// TIA Portal V18 export
FUNCTION_BLOCK "LAxisGroupBasics_AxisGroupBasics_Grp1"   // FB5, SCL
{ S7_Optimized_Access := 'TRUE' }
// stored: MemoryReserve 100, SetENOAutomatically false
   VAR_INPUT
      powerEnableAll : Bool;   // MC_Power: 0: Disable all axes/ 1: Enable all axes
      homeExecuteAll : Bool;   // MC_Home: Start job for all axes with positive edge
      resetExecuteAll : Bool;   // MC_Reset: Start job for all axes with positive edge
      restartAll : Bool;   // 0: Acknowledgment of queued technology alarms / 1: Reinitialization of the technology object and acknowledgment of pending technology alarms
      haltExecuteAll : Bool;   // MC_Halt: Start job for all axes with positive edge
   END_VAR
   VAR_OUTPUT
      powerStatusGroup : Bool;   // MC_Power: 0: At least one Technology object disabled / 1: All Technology objects enabled
      homingStatusGroup : Bool;   // MC_Home: 0: At least one Technology object
      busy : Bool;   // Job is running
      done : Bool;   // All active jobs done
      commandAborted : Bool;   // At least one command was aborted
      error : Bool;   // An error occurred during execution of the job. The job is rejected. The cause of the error can be found in the "Status" parameter.
      status : Word;   // Status information
      diagnostics : "LAxisGroupBasics_typeDiagnostics";   // Diagnostics information
   END_VAR
   VAR_IN_OUT
      axisGroupBasicsData : Array[*] of "LAxisGroupBasics_typeAxisGroupBasicsData";   // Axis data
   END_VAR
   VAR
      instAxisBasics : Array[#LOWER_LIMIT_AXES_ARRAY..#UPPER_LIMIT_AXES_ARRAY] of "LAxisBasics_AxisBasics";
      statErrorIndexOld { ExternalAccessible := 'False'; ExternalVisible := 'False'; ExternalWritable := 'False'} : DInt;   // Flag for saving error index
      statAxisBasicsStatusOld { ExternalAccessible := 'False'; ExternalVisible := 'False'; ExternalWritable := 'False'} : Word;   // Flag for saving LAxisBasics status
      statAxisBasicsSubfunctionStatusOld { ExternalAccessible := 'False'; ExternalVisible := 'False'; ExternalWritable := 'False'} : Word;   // Flag for savin LAxisBasics subfunction status
   END_VAR
   VAR_TEMP
      tempAxisArrayLowerBound : DInt;   // Start index of axes array
      tempAxisArrayUpperBound : DInt;   // End index of axes array
      tempIndex : DInt;   // index counter
      tempDateTimeRetVal : Int;   // date time return value
      tempError : Bool;   // temporary error bit
      tempBusy : Bool;   // temporary busy bit
      tempDone : Bool;   // temporary done bit
      tempCmdAborted : Bool;   // temporary command aborted bit
      tempPowerStatusGroup : Bool;   // temporary power status group bit
      tempHomingStatusGroup : Bool;   // temporary homing status group bit
      tempFirstErrorIndex : DInt;   // index at which first error occured
      tempNewError : Bool;   // new error occured in this cycle
   END_VAR
   VAR CONSTANT
      LOWER_LIMIT_AXES_ARRAY : DInt := 0;   // Start index of axes array needs to be adapted to real array dimensons
      UPPER_LIMIT_AXES_ARRAY : DInt := 4;   // End index of axes array needs to be adapted to real array dimensions
      STATUS_INCORRECT_ARRAY_CONSTANTS : Word := 16#8310;   // status value incorrect array constants
      STATUS_ERR_SYSTEMFUNCTION : Word := 16#8600;   // status value error LAxisBasics
      STATUS_ACTIVE : Word := 16#7002;   // status value active
      STATUS_INACTIVE : Word := 16#7000;   // status value inactive
      DEFAULT_DATE_TIME : Date_And_Time := DT#1990-01-01-00:00:00;   // date and time default value
      DEFAULT_STATUS : Word := 16#0;   // status value default
      ADD_VALUE1_DEFAULT : Int := 0;   // additional value 1 default
      ADD_VALUE2_DEFAULT : Word;   // additional value 2 default
      EMPTY : DInt := -1;   // empty
   END_VAR
BEGIN
   //=============================================================================
   //SIEMENS AG
   //(c)Copyright 2016 All Rights Reserved
   //-----------------------------------------------------------------------------
   //Library:       Axis Basics
   //Tested with:   S7-1500T V3.0
   //Engineering:   TIA Portal V18
   //Restrictions:  Motion Control Library V7.0
   //Requirements:  S7-1500(T)
   //Functionality: Basic axis group control and data collection
   //-----------------------------------------------------------------------------
   //Change log table:
   //Version  Date       Expert in charge Changes applied
   //01.00.00 01.08.2023 FrJu             First released version
   //=============================================================================

   REGION Axis array checks
       //Check Array boundaries of axis array
       #tempAxisArrayUpperBound := UPPER_BOUND(ARR := #axisGroupBasicsData, DIM := 1);
       #tempAxisArrayLowerBound := LOWER_BOUND(ARR := #axisGroupBasicsData, DIM := 1);

       //Check if number of axes/array length is matching - output error and return if values are not matching
       IF #tempAxisArrayUpperBound <> #UPPER_LIMIT_AXES_ARRAY
           OR #tempAxisArrayLowerBound <> #LOWER_LIMIT_AXES_ARRAY THEN

           #error := TRUE;
           #status := #diagnostics.status := #STATUS_INCORRECT_ARRAY_CONSTANTS;

           RETURN;
       END_IF;
   END_REGION

   REGION Initialize values
       //initialize values
       #tempError := FALSE;
       #tempBusy := FALSE;
       #tempDone := FALSE;
       #tempPowerStatusGroup := TRUE;
       #tempHomingStatusGroup := TRUE;
       #tempFirstErrorIndex := #EMPTY;
       #tempCmdAborted := FAlSE;
   END_REGION

   REGION Axes operation loop
       //Loop through all instances of LAxisBasics and execute commands
       FOR #tempIndex := #tempAxisArrayLowerBound TO #tempAxisArrayUpperBound DO

           REGION Call AxisBasics
               //Call LAxisBasics_AxisBasics
               #instAxisBasics[#tempIndex](axis := #axisGroupBasicsData[#tempIndex].axis,
                                           powerEnable := #axisGroupBasicsData[#tempIndex].axisBasicsData.axisControl.axisControlCommand.powerEnable OR #powerEnableAll,
                                           powerStartMode := #axisGroupBasicsData[#tempIndex].axisBasicsData.axisControl.axisControlCommand.powerStartMode,
                                           powerStopMode := #axisGroupBasicsData[#tempIndex].axisBasicsData.axisControl.axisControlCommand.powerStopMode,
                                           resetExecute := #axisGroupBasicsData[#tempIndex].axisBasicsData.axisControl.axisControlCommand.resetExecute OR #resetExecuteAll,
                                           resetRestart := #axisGroupBasicsData[#tempIndex].axisBasicsData.axisControl.axisControlCommand.resetRestart OR #restartAll,
                                           homeExecute := #axisGroupBasicsData[#tempIndex].axisBasicsData.axisControl.axisControlCommand.homeExecute OR #homeExecuteAll,
                                           homePosition := #axisGroupBasicsData[#tempIndex].axisBasicsData.axisControl.axisControlCommand.homePosition,
                                           homeMode := #axisGroupBasicsData[#tempIndex].axisBasicsData.axisControl.axisControlCommand.homeMode,
                                           jogForward := #axisGroupBasicsData[#tempIndex].axisBasicsData.axisControl.axisControlCommand.jogForward,
                                           jogBackward := #axisGroupBasicsData[#tempIndex].axisBasicsData.axisControl.axisControlCommand.jogBackward,
                                           jogVelocity := #axisGroupBasicsData[#tempIndex].axisBasicsData.axisControl.axisControlCommand.jogVelocity,
                                           jogAcceleration := #axisGroupBasicsData[#tempIndex].axisBasicsData.axisControl.axisControlCommand.jogAcceleration,
                                           jogDeceleration := #axisGroupBasicsData[#tempIndex].axisBasicsData.axisControl.axisControlCommand.jogDeceleration,
                                           jogJerk := #axisGroupBasicsData[#tempIndex].axisBasicsData.axisControl.axisControlCommand.jogJerk,
                                           jogPositionControlled := #axisGroupBasicsData[#tempIndex].axisBasicsData.axisControl.axisControlCommand.jogPositionControlled,
                                           moveAbsExecute := #axisGroupBasicsData[#tempIndex].axisBasicsData.axisControl.axisControlCommand.moveAbsExecute,
                                           moveRelExecute := #axisGroupBasicsData[#tempIndex].axisBasicsData.axisControl.axisControlCommand.moveRelExecute,
                                           movePosition := #axisGroupBasicsData[#tempIndex].axisBasicsData.axisControl.axisControlCommand.movePosition,
                                           moveDistance := #axisGroupBasicsData[#tempIndex].axisBasicsData.axisControl.axisControlCommand.moveDistance,
                                           moveVelocity := #axisGroupBasicsData[#tempIndex].axisBasicsData.axisControl.axisControlCommand.moveVelocity,
                                           moveAcceleration := #axisGroupBasicsData[#tempIndex].axisBasicsData.axisControl.axisControlCommand.moveAcceleration,
                                           moveDeceleration := #axisGroupBasicsData[#tempIndex].axisBasicsData.axisControl.axisControlCommand.moveDeceleration,
                                           moveJerk := #axisGroupBasicsData[#tempIndex].axisBasicsData.axisControl.axisControlCommand.moveJerk,
                                           moveDirection := #axisGroupBasicsData[#tempIndex].axisBasicsData.axisControl.axisControlCommand.moveDirection,
                                           haltExecute := #axisGroupBasicsData[#tempIndex].axisBasicsData.axisControl.axisControlCommand.haltExecute OR #haltExecuteAll,
                                           haltDeceleration := #axisGroupBasicsData[#tempIndex].axisBasicsData.axisControl.axisControlCommand.haltDeceleration,
                                           haltJerk := #axisGroupBasicsData[#tempIndex].axisBasicsData.axisControl.axisControlCommand.haltJerk,
                                           haltAbortAcceleration := #axisGroupBasicsData[#tempIndex].axisBasicsData.axisControl.axisControlCommand.haltAbortAcceleration,
                                           axisDataConfig := #axisGroupBasicsData[#tempIndex].axisBasicsData.axisData.axisDataConfig,
                                           powerStatus => #axisGroupBasicsData[#tempIndex].axisBasicsData.axisControl.axisControlStatus.powerStatus,
                                           powerBusy => #axisGroupBasicsData[#tempIndex].axisBasicsData.axisControl.axisControlStatus.powerBusy,
                                           resetDone => #axisGroupBasicsData[#tempIndex].axisBasicsData.axisControl.axisControlStatus.resetDone,
                                           resetBusy => #axisGroupBasicsData[#tempIndex].axisBasicsData.axisControl.axisControlStatus.resetBusy,
                                           homeDone => #axisGroupBasicsData[#tempIndex].axisBasicsData.axisControl.axisControlStatus.homeDone,
                                           homeBusy => #axisGroupBasicsData[#tempIndex].axisBasicsData.axisControl.axisControlStatus.homeBusy,
                                           jogInVelocity => #axisGroupBasicsData[#tempIndex].axisBasicsData.axisControl.axisControlStatus.jogInVelocity,
                                           jogBusy => #axisGroupBasicsData[#tempIndex].axisBasicsData.axisControl.axisControlStatus.jogBusy,
                                           moveAbsDone => #axisGroupBasicsData[#tempIndex].axisBasicsData.axisControl.axisControlStatus.moveAbsDone,
                                           moveAbsBusy => #axisGroupBasicsData[#tempIndex].axisBasicsData.axisControl.axisControlStatus.moveAbsBusy,
                                           moveRelDone => #axisGroupBasicsData[#tempIndex].axisBasicsData.axisControl.axisControlStatus.moveRelDone,
                                           moveRelBusy => #axisGroupBasicsData[#tempIndex].axisBasicsData.axisControl.axisControlStatus.moveRelBusy,
                                           haltDone => #axisGroupBasicsData[#tempIndex].axisBasicsData.axisControl.axisControlStatus.haltDone,
                                           haltBusy => #axisGroupBasicsData[#tempIndex].axisBasicsData.axisControl.axisControlStatus.haltBusy,
                                           commandAborted => #axisGroupBasicsData[#tempIndex].axisBasicsData.axisControl.axisControlStatus.commandAborted,
                                           error => #axisGroupBasicsData[#tempIndex].axisBasicsData.axisControl.axisControlStatus.error,
                                           status => #axisGroupBasicsData[#tempIndex].axisBasicsData.axisControl.axisControlStatus.status,
                                           diagnostics => #axisGroupBasicsData[#tempIndex].axisBasicsData.axisControl.axisControlStatus.diagnostics,
                                           axisData => #axisGroupBasicsData[#tempIndex].axisBasicsData.axisData.axisDataValues);
           END_REGION



           REGION Status values
               //set error and status if at least one instance of AxisBasics shows an error
               IF #axisGroupBasicsData[#tempIndex].axisBasicsData.axisControl.axisControlStatus.error THEN
                   #tempError := true;
                   #tempDone := false;
                   IF #tempFirstErrorIndex = #EMPTY THEN
                       #tempFirstErrorIndex := #tempIndex;
                   END_IF;
               END_IF;

               //Reset axes group homing status if at least one axis is not homed
               IF NOT #axisGroupBasicsData[#tempIndex].axisBasicsData.axisData.axisDataValues.axisStatus.statusWord.bit05_HomingDone THEN
                   #tempHomingStatusGroup := FALSE;
               END_IF;

               //Reset group power status if at least one axis is not powered on
               IF NOT #axisGroupBasicsData[#tempIndex].axisBasicsData.axisControl.axisControlStatus.powerStatus THEN
                   #tempPowerStatusGroup := FALSE;
               END_IF;

               //set busy output if at least one instance of AxisBasics is busy
               IF #axisGroupBasicsData[#tempIndex].axisBasicsData.axisControl.axisControlStatus.resetBusy
                   OR #axisGroupBasicsData[#tempIndex].axisBasicsData.axisControl.axisControlStatus.homeBusy
                   OR #axisGroupBasicsData[#tempIndex].axisBasicsData.axisControl.axisControlStatus.jogBusy
                   OR #axisGroupBasicsData[#tempIndex].axisBasicsData.axisControl.axisControlStatus.moveAbsBusy
                   OR #axisGroupBasicsData[#tempIndex].axisBasicsData.axisControl.axisControlStatus.moveRelBusy
                   OR #axisGroupBasicsData[#tempIndex].axisBasicsData.axisControl.axisControlStatus.haltBusy
               THEN
                   #tempBusy := true;
               END_IF;

               //set command aborted if at least one command was aborted
               IF #axisGroupBasicsData[#tempIndex].axisBasicsData.axisControl.axisControlStatus.commandAborted THEN
                   #tempCmdAborted := true;
               END_IF;

               //Set done for Group commands
               IF NOT #tempBusy AND NOT #tempError AND NOT #tempCmdAborted AND
                   (#axisGroupBasicsData[#tempIndex].axisBasicsData.axisControl.axisControlStatus.homeDone OR
                   #axisGroupBasicsData[#tempIndex].axisBasicsData.axisControl.axisControlStatus.resetDone OR
                   #axisGroupBasicsData[#tempIndex].axisBasicsData.axisControl.axisControlStatus.haltDone OR
                   #axisGroupBasicsData[#tempIndex].axisBasicsData.axisControl.axisControlStatus.moveAbsDone OR
                   #axisGroupBasicsData[#tempIndex].axisBasicsData.axisControl.axisControlStatus.moveRelDone)
               THEN
                   #tempDone := TRUE;
               END_IF;
           END_REGION
       END_FOR;
   END_REGION

   REGION Status
       //set status output
       IF #tempError THEN
           #status := #diagnostics.status := #STATUS_ERR_SYSTEMFUNCTION;
       ELSIF #tempBusy THEN
           #status := #diagnostics.status := #STATUS_ACTIVE;
       ELSE
           #status := #diagnostics.status := #STATUS_INACTIVE;
       END_IF;

   END_REGION

   REGION Set output values
       #busy := #tempBusy;
       #done := #tempDone;
       #powerStatusGroup := #tempPowerStatusGroup;
       #homingStatusGroup := #tempHomingStatusGroup;
       #commandAborted := #tempCmdAborted;


       //Check if new error occured in this cycle
       IF #tempFirstErrorIndex <= #UPPER_LIMIT_AXES_ARRAY
           AND #tempFirstErrorIndex >= #LOWER_LIMIT_AXES_ARRAY
       THEN
           IF #statErrorIndexOld <> #tempFirstErrorIndex
               OR #statAxisBasicsStatusOld <> #axisGroupBasicsData[#tempFirstErrorIndex].axisBasicsData.axisControl.axisControlStatus.status
               OR #statAxisBasicsSubfunctionStatusOld <> #axisGroupBasicsData[#tempFirstErrorIndex].axisBasicsData.axisControl.axisControlStatus.diagnostics.subFunctionStatus
           THEN
               #tempNewError := TRUE;
           END_IF;
       END_IF;

       //Save actual error information for next cycle
       #statErrorIndexOld := #tempFirstErrorIndex;
       IF #tempFirstErrorIndex <= #UPPER_LIMIT_AXES_ARRAY
           AND #tempFirstErrorIndex >= #LOWER_LIMIT_AXES_ARRAY THEN
           #statAxisBasicsStatusOld := #axisGroupBasicsData[#tempFirstErrorIndex].axisBasicsData.axisControl.axisControlStatus.status;
           #statAxisBasicsSubfunctionStatusOld := #axisGroupBasicsData[#tempFirstErrorIndex].axisBasicsData.axisControl.axisControlStatus.diagnostics.subFunctionStatus;
       ELSE
           #statAxisBasicsStatusOld := #DEFAULT_STATUS;
           #statAxisBasicsSubfunctionStatusOld := #DEFAULT_STATUS;
       END_IF;

       //Set diagnostics values if new error occured
       IF #tempError THEN
           IF #tempNewError THEN
               #error := true;
               #tempDateTimeRetVal := RD_LOC_T(#diagnostics.timestamp);
               #diagnostics.additionalValue1 := #tempFirstErrorIndex;
               IF #tempFirstErrorIndex <= #UPPER_LIMIT_AXES_ARRAY
                   AND #tempFirstErrorIndex >= #LOWER_LIMIT_AXES_ARRAY
               THEN
                   #diagnostics.additionalValue2 := #axisGroupBasicsData[#tempFirstErrorIndex].axisBasicsData.axisControl.axisControlStatus.diagnostics.subFunctionStatus;
                   #diagnostics.subFunctionStatus := #axisGroupBasicsData[#tempFirstErrorIndex].axisBasicsData.axisControl.axisControlStatus.status;
               END_IF;
           END_IF;
       ELSE
           //reset error information if no error occured in this cycle
           #error := false;
           #diagnostics.subFunctionStatus := #DEFAULT_STATUS;
           #diagnostics.additionalValue1 := #ADD_VALUE1_DEFAULT;
           #diagnostics.additionalValue2 := #ADD_VALUE2_DEFAULT;
           #diagnostics.timestamp := #DEFAULT_DATE_TIME;
       END_IF;
   END_REGION
END_FUNCTION_BLOCK
